// TIA Portal V20 export
DATA_BLOCK "CMInterface_Dosing_DB"   // DB27
// stored: InstanceOfName CM_Interface_Dosing, InstanceOfType FB
"CM_Interface_Dosing"
   // VAR_INPUT
   //    CmCommand { ExternalAccessible := 'False'; ExternalVisible := 'False'; ExternalWritable := 'False'} : Array[0..29] of Bool;
   //    Procedure_Param { ExternalAccessible := 'False'; ExternalVisible := 'False'; ExternalWritable := 'False'} : Array[0..31] of Real;
   //    CmFbOnOff { ExternalAccessible := 'False'; ExternalVisible := 'False'; ExternalWritable := 'False'} : Array[0..29] of Bool;
   //    Pumped_Liters : Real;
   //    Auto_Man : Bool;
   //    Oos : Bool;
   // END_VAR
   // VAR_OUTPUT
   //    CM_P100 { ExternalAccessible := 'False'; ExternalVisible := 'False'; ExternalWritable := 'False'} : "DigVal";
   //    CM_V102 { ExternalAccessible := 'False'; ExternalVisible := 'False'; ExternalWritable := 'False'} : "DigVal";
   //    CM_V103 { ExternalAccessible := 'False'; ExternalVisible := 'False'; ExternalWritable := 'False'} : "DigVal";
   //    CM_V104 { ExternalAccessible := 'False'; ExternalVisible := 'False'; ExternalWritable := 'False'} : "DigVal";
   //    QuantityProduct { ExternalAccessible := 'False'; ExternalVisible := 'False'; ExternalWritable := 'False'} : "AnaVal";
   // END_VAR
   // VAR
   //    Pos_edge : Bool;
   //    Neg_edge : Bool;
   // END_VAR
BEGIN
END_DATA_BLOCK
